Yaskawa INFORM job: small_flange_cylinder_program.JBI

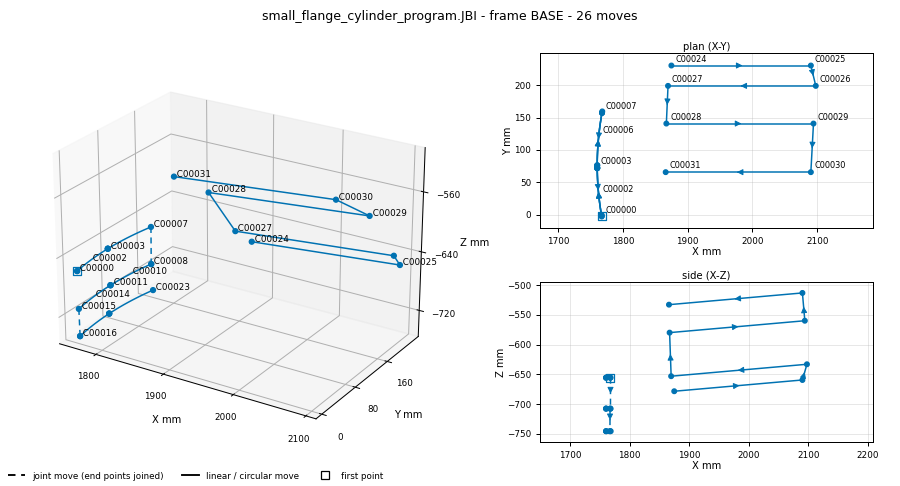
[picture p0: tool path of small_flange_cylinder_program.JBI in frame BASE, 26 of 37 moves have a stored position in this frame; points joined in program order, loops and branches not executed]
/JOB
//NAME small_flange_cylinder_program
//POS
///NPOS 32,0,32,0,0,0
///TOOL 0
///POSTYPE BASE
///RECTAN
///RCONF 0,0,0,0,0,0,0,0,0,0,0,0,0,0,0,0,0,0,0,0,0,0,0,0
C00000=1767.276163,-2.462911,-655.432960,175.000000,-60.000000,10.049761
C00001=1767.276163,-2.462911,-655.432960,175.000000,-60.000000,10.049761
C00002=1762.731748,30.037670,-655.432960,175.000000,-60.000000,5.869862
C00003=1760.386442,72.526856,-655.432960,-175.000000,-60.000000,5.000000
C00004=1760.386442,72.526856,-655.432960,-175.000000,-60.000000,5.000000
C00005=1760.386442,72.526856,-655.432960,-175.000000,-60.000000,5.000000
C00006=1762.527564,120.035178,-655.432960,-175.000000,-60.000000,-5.609879
C00007=1767.874428,157.871105,-655.432960,175.000000,-60.000000,-10.477342
C00008=1767.744902,157.167577,-707.415960,-175.000000,-60.000000,-10.386247
C00009=1767.744902,157.167577,-707.415960,-175.000000,-60.000000,-10.386247
C00010=1762.261859,117.240520,-707.415960,175.000000,-60.000000,-5.252395
C00011=1760.372708,76.313027,-707.415960,-175.000000,-60.000000,-5.000000
C00012=1760.372708,76.313027,-707.415960,-175.000000,-60.000000,-5.000000
C00013=1760.372708,76.313027,-707.415960,-175.000000,-60.000000,-5.000000
C00014=1762.147701,36.124955,-707.415960,175.000000,-60.000000,5.091125
C00015=1767.047862,-1.163618,-707.415960,175.000000,-60.000000,9.881770
C00016=1766.880717,-0.197895,-745.356460,175.000000,-60.000000,9.756964
C00017=1766.880717,-0.197895,-745.356460,175.000000,-60.000000,9.756964
C00018=1763.011587,27.392604,-745.356460,175.000000,-60.000000,6.208572
C00019=1760.392388,71.835747,-745.356460,-175.000000,-60.000000,5.000000
C00020=1760.392388,71.835747,-745.356460,-175.000000,-60.000000,5.000000
C00021=1760.392388,71.835747,-745.356460,-175.000000,-60.000000,5.000000
C00022=1763.151058,125.977023,-745.356460,-175.000000,-60.000000,-6.370689
C00023=1768.190923,159.564404,-745.356460,175.000000,-60.000000,-10.696705
C00024=1874.898891,230.423665,-678.229476,175.000000,-60.000000,-89.314857
C00025=2090.243281,230.423689,-659.299066,175.000000,-60.000000,-89.314857
C00026=2097.824131,199.011992,-632.908554,-175.000000,-61.636461,-87.279760
C00027=1869.705391,199.011966,-652.961926,-175.000000,-61.636461,-87.279760
C00028=1867.102606,140.810568,-579.750435,-175.000000,-41.722893,-84.342242
C00029=2094.283827,140.810594,-559.779478,-175.000000,-41.722893,-84.342242
C00030=2090.232165,65.778953,-513.077639,157.338074,-5.000000,5.000000
C00031=1866.073357,65.778927,-532.782904,157.338074,-5.000000,5.000000
///POSTYPE PULSE
///PULSE
EX00000=144384.0
EX00001=334848.0
///POSTYPE PULSE
///PULSE
EC00000=144384.0
EC00001=144384.0
EC00002=144384.0
EC00003=144384.0
EC00004=144384.0
EC00005=144384.0
EC00006=144384.0
EC00007=144384.0
EC00008=144384.0
EC00009=144384.0
EC00010=144384.0
EC00011=144384.0
EC00012=144384.0
EC00013=144384.0
EC00014=144384.0
EC00015=144384.0
EC00016=144384.0
EC00017=144384.0
EC00018=144384.0
EC00019=144384.0
EC00020=144384.0
EC00021=144384.0
EC00022=144384.0
EC00023=144384.0
EC00024=334848.0
EC00025=334848.0
EC00026=334848.0
EC00027=334848.0
EC00028=334848.0
EC00029=334848.0
EC00030=334848.0
EC00031=334848.0
//INST
///DATE 2023/08/16 15:56
///ATTR SC,RW,RJ
////FRAME BASE
///GROUP1 RB1,ST1
NOP
MOVJ P009 EX000 VJ=15.00
MOVJ C00000 EC00000 VJ=15.0
CALL JOB:SPYON
MOVC C00001 EC00001 V=150.0
MOVC C00002 EC00002 V=150.0
MOVC C00003 EC00003 V=150.0
MOVJ C00004 EC00004 VJ=15.0
MOVC C00005 EC00005 V=150.0
MOVC C00006 EC00006 V=150.0
MOVC C00007 EC00007 V=150.0
MOVJ C00008 EC00008 VJ=15.0
MOVC C00009 EC00009 V=150.0
MOVC C00010 EC00010 V=150.0
MOVC C00011 EC00011 V=150.0
MOVJ C00012 EC00012 VJ=15.0
MOVC C00013 EC00013 V=150.0
MOVC C00014 EC00014 V=150.0
MOVC C00015 EC00015 V=150.0
MOVJ C00016 EC00016 VJ=15.0
MOVC C00017 EC00017 V=150.0
MOVC C00018 EC00018 V=150.0
MOVC C00019 EC00019 V=150.0
MOVJ C00020 EC00020 VJ=15.0
MOVC C00021 EC00021 V=150.0
MOVC C00022 EC00022 V=150.0
MOVC C00023 EC00023 V=150.0
CALL JOB:SPYOF
MOVJ P009 VJ=15.00
MOVL P009 EX00000 V=150.0
MOVJ C00024 EC00024 VJ=15.0
CALL JOB:SPYON
MOVL C00025 EC00025 V=150.0
MOVL C00026 EC00026 V=150.0
MOVL C00027 EC00027 V=150.0
MOVL C00028 EC00028 V=150.0
MOVL C00029 EC00029 V=150.0
MOVL C00030 EC00030 V=150.0
MOVL C00031 EC00031 V=150.0
CALL JOB:SPYOF
MOVJ P009 VJ=15.00
MOVL P009 EX00001 V=150.0
END
